PROGRAM GL10_Transfer_Traverse
VAR
	GL10: sTransfer;
	GL11: sTransfer;
	GL12: sTransfer;
	GL3: sConveyor;
	GL7: sConveyor;
	GL9: sConveyor;
	GL10_RD: SRoll_Door;
	GL12_RD: SRoll_Door;
	RUN_FWD_TO_GL3_BIT : BOOL; // GL11 OCCUPIED, GL3 REQUESTING PART, RUN TO GL3 POSITION
	RUN_REV_TO_GL7_BIT : BOOL; // GL11 EMPTY, GL7 REQUESTING PICK UP, RUN TO GL7 POSITION
	RUN_REV_TO_GL9_BIT : BOOL; // GL11 EMPTY, GL9 REQUESTING PICK UP, RUN TO GL9 POSITION
	RUN_REV_TO_GL12_BIT : BOOL; // GL11 EMPTY, GL11 RUN TO GL12 POSITION
END_VAR
VAR // added by the converter: edge detectors and wires of the graphical bodies
    _w1 : BOOL;
END_VAR

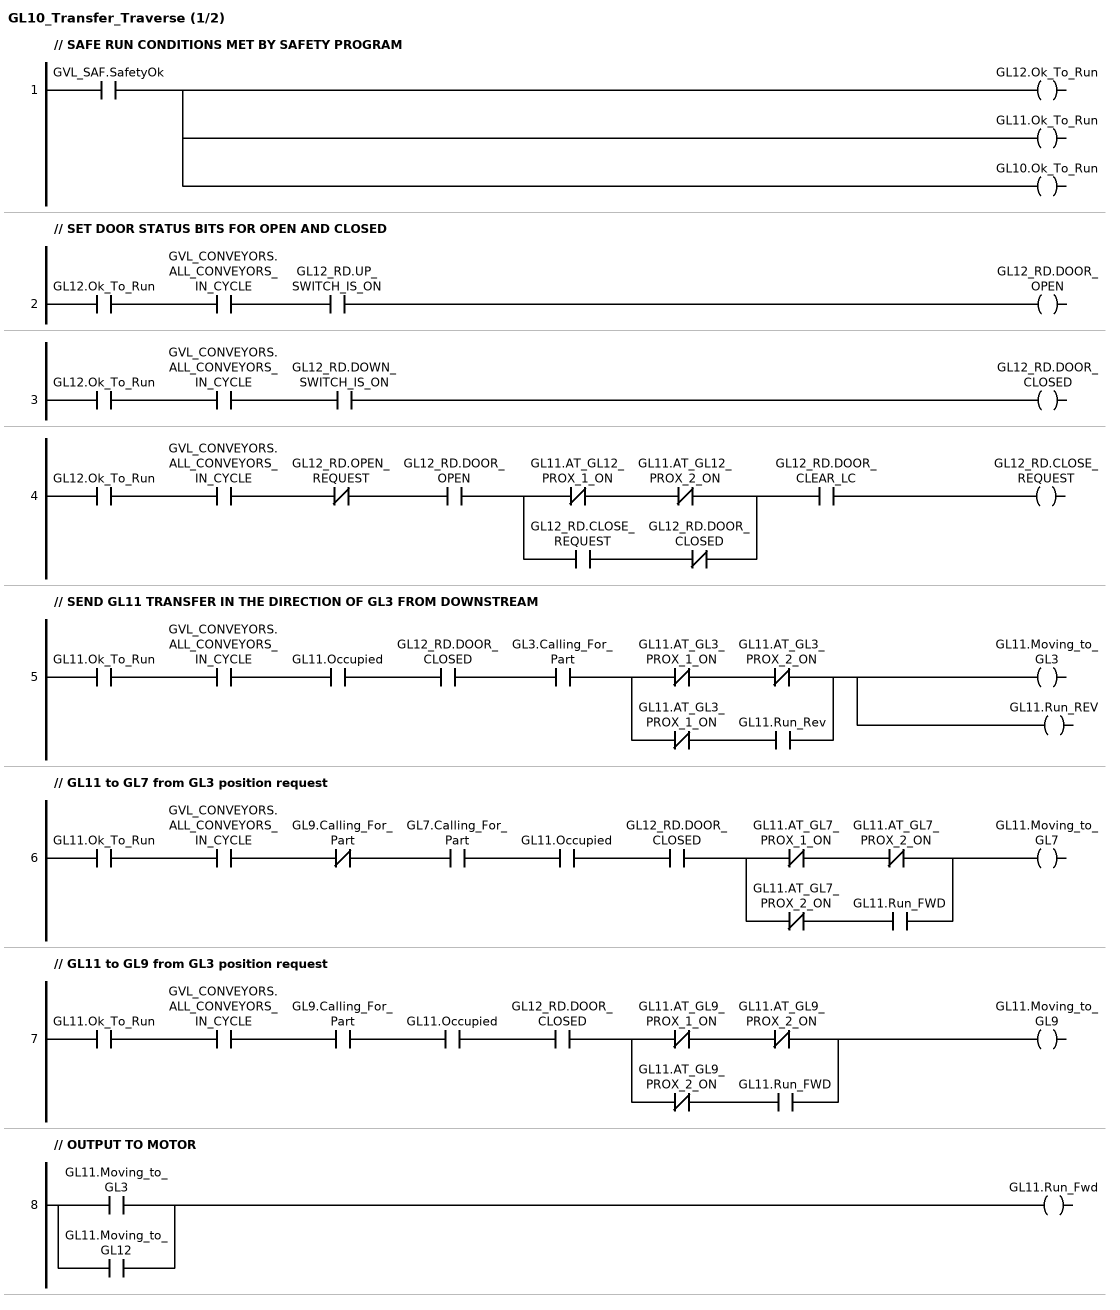
// NETWORK 1: // SAFE RUN CONDITIONS MET BY SAFETY PROGRAM
GL12.Ok_To_Run := GVL_SAF.SafetyOk;
GL11.Ok_To_Run := GVL_SAF.SafetyOk;
GL10.Ok_To_Run := GVL_SAF.SafetyOk;

// NETWORK 2: // SET DOOR STATUS BITS FOR OPEN AND CLOSED
GL12_RD.DOOR_OPEN := GL12.Ok_To_Run AND GVL_CONVEYORS.ALL_CONVEYORS_IN_CYCLE AND GL12_RD.UP_SWITCH_IS_ON;

// NETWORK 3
GL12_RD.DOOR_CLOSED := GL12.Ok_To_Run AND GVL_CONVEYORS.ALL_CONVEYORS_IN_CYCLE AND GL12_RD.DOWN_SWITCH_IS_ON;

// NETWORK 4
GL12_RD.CLOSE_REQUEST := GL12.Ok_To_Run AND GVL_CONVEYORS.ALL_CONVEYORS_IN_CYCLE AND NOT GL12_RD.OPEN_REQUEST AND GL12_RD.DOOR_OPEN AND (NOT GL11.AT_GL12_PROX_1_ON AND NOT GL11.AT_GL12_PROX_2_ON OR GL12_RD.CLOSE_REQUEST AND NOT GL12_RD.DOOR_CLOSED) AND GL12_RD.DOOR_CLEAR_LC;

// NETWORK 5: // SEND GL11 TRANSFER IN THE DIRECTION OF GL3 FROM DOWNSTREAM
_w1 := GL11.Ok_To_Run AND GVL_CONVEYORS.ALL_CONVEYORS_IN_CYCLE AND GL11.Occupied AND GL12_RD.DOOR_CLOSED AND GL3.Calling_For_Part AND (NOT GL11.AT_GL3_PROX_1_ON AND NOT GL11.AT_GL3_PROX_2_ON OR NOT GL11.AT_GL3_PROX_1_ON AND GL11.Run_Rev);
GL11.Moving_to_GL3 := _w1;
GL11.Run_REV := _w1;

// NETWORK 6: // GL11 to GL7 from GL3 position request
GL11.Moving_to_GL7 := GL11.Ok_To_Run AND GVL_CONVEYORS.ALL_CONVEYORS_IN_CYCLE AND NOT GL9.Calling_For_Part AND GL7.Calling_For_Part AND GL11.Occupied AND GL12_RD.DOOR_CLOSED AND (NOT GL11.AT_GL7_PROX_1_ON AND NOT GL11.AT_GL7_PROX_2_ON OR NOT GL11.AT_GL7_PROX_2_ON AND GL11.Run_FWD);

// NETWORK 7: // GL11 to GL9 from GL3 position request
GL11.Moving_to_GL9 := GL11.Ok_To_Run AND GVL_CONVEYORS.ALL_CONVEYORS_IN_CYCLE AND GL9.Calling_For_Part AND GL11.Occupied AND GL12_RD.DOOR_CLOSED AND (NOT GL11.AT_GL9_PROX_1_ON AND NOT GL11.AT_GL9_PROX_2_ON OR NOT GL11.AT_GL9_PROX_2_ON AND GL11.Run_FWD);

// NETWORK 8: // OUTPUT TO MOTOR
GL11.Run_Fwd := GL11.Moving_to_GL3 OR GL11.Moving_to_GL12;

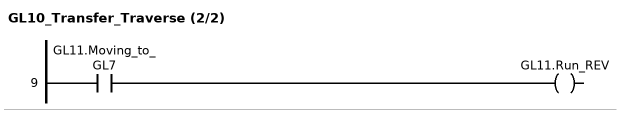
// NETWORK 9
GL11.Run_REV := GL11.Moving_to_GL7;

END_PROGRAM

(* stored: Version 1.1.0.1, ProductVersion 3.1.4024.12
   POU GL10_Transfer_Traverse: Id {007c7d62-b5d8-4adc-addb-9b40e59320f7}, SpecialFunc None *)
